// LS Electric XG5000 project: 과년68_2_3
// PLC NewPLC
// module base 0 slot 0: 입출력 모듈:XBC-DR20S (DC 24V 입력 12점, 릴레이 출력 8점)

PROGRAM NewProgram (task: 스캔 프로그램)

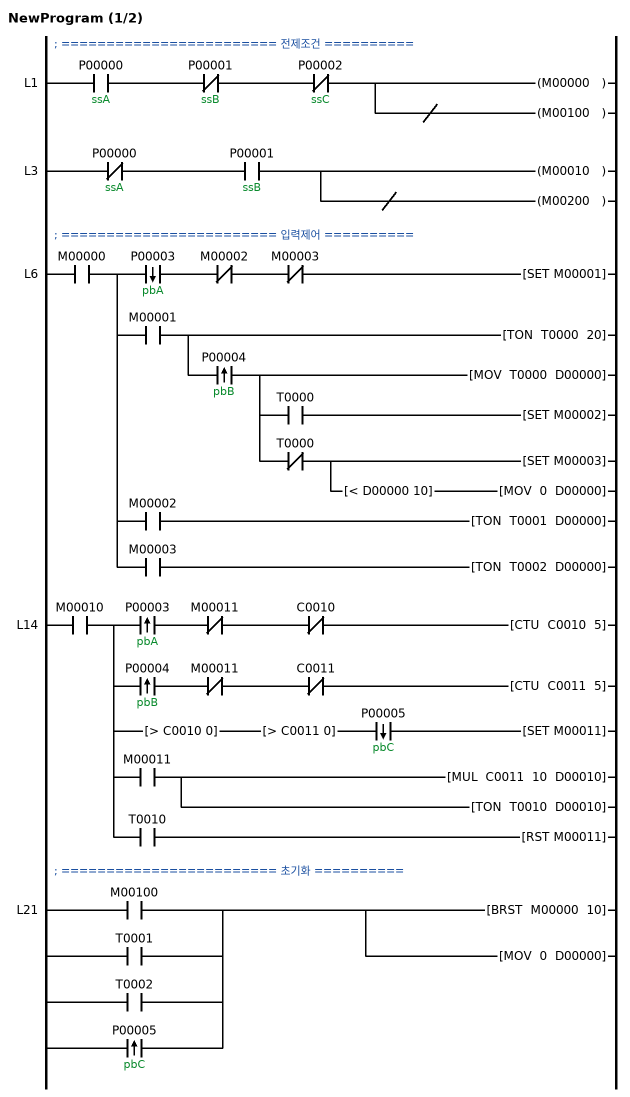
// ======================== 전제조건 ==========
; L1
LOAD      P00000	// ssA
AND NOT   P00001	// ssB
AND NOT   P00002	// ssC
OUT       M00000
NOT
OUT       M00100
; L3
LOAD NOT  P00000	// ssA
AND       P00001	// ssB
OUT       M00010
NOT
OUT       M00200
// ======================== 입력제어 ==========
; L6
LOAD      M00000
MPUSH
ANDN      P00003	// pbA
AND NOT   M00002
AND NOT   M00003
SET       M00001
MLOAD
AND       M00001
TON       T0000 20
ANDP      P00004	// pbB
MOV       T0000 D00000
MPUSH
AND       T0000
SET       M00002
MPOP
AND NOT   T0000
SET       M00003
AND<      D00000 10
MOV       0 D00000
MLOAD
AND       M00002
TON       T0001 D00000
MPOP
AND       M00003
TON       T0002 D00000
; L14
LOAD      M00010
MPUSH
ANDP      P00003	// pbA
AND NOT   M00011
AND NOT   C0010
CTU       C0010 5
MLOAD
ANDP      P00004	// pbB
AND NOT   M00011
AND NOT   C0011
CTU       C0011 5
MLOAD
AND>      C0010 0
AND>      C0011 0
ANDN      P00005	// pbC
SET       M00011
MLOAD
AND       M00011
MUL       C0011 10 D00010
TON       T0010 D00010
MPOP
AND       T0010
RST       M00011
// ======================== 초기화 ==========
; L21
LOAD      M00100
OR        T0001
OR        T0002
ORP       P00005	// pbC
BRST      M00000 10
MOV       0 D00000

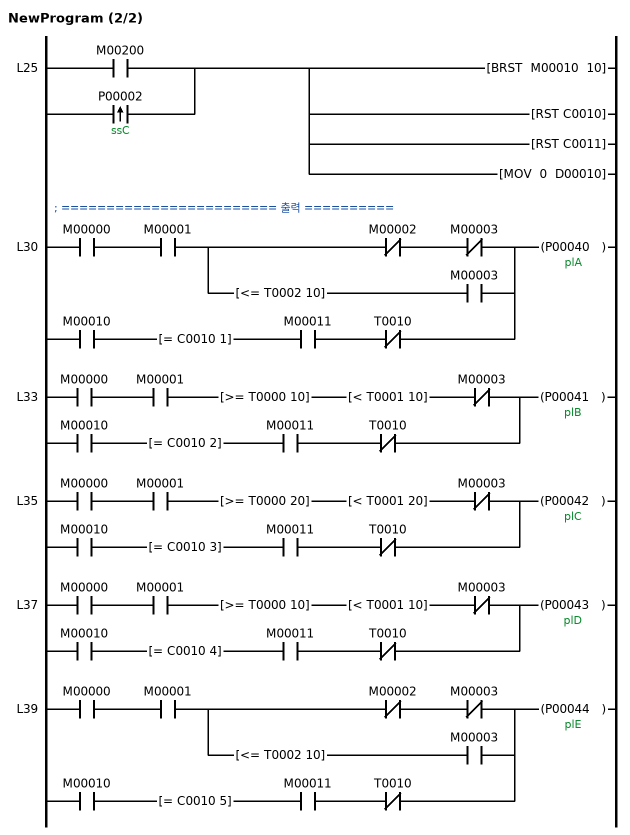
; L25
LOAD      M00200
ORP       P00002	// ssC
BRST      M00010 10
RST       C0010
RST       C0011
MOV       0 D00010
// ======================== 출력 ==========
; L30
LOAD      M00000
AND       M00001
LOAD NOT  M00002
AND NOT   M00003
LOAD<=    T0002 10
AND       M00003
OR LOAD
AND LOAD
LOAD      M00010
AND=      C0010 1
AND       M00011
AND NOT   T0010
OR LOAD
OUT       P00040	// plA
; L33
LOAD      M00000
AND       M00001
AND>=     T0000 10
AND<      T0001 10
AND NOT   M00003
LOAD      M00010
AND=      C0010 2
AND       M00011
AND NOT   T0010
OR LOAD
OUT       P00041	// plB
; L35
LOAD      M00000
AND       M00001
AND>=     T0000 20
AND<      T0001 20
AND NOT   M00003
LOAD      M00010
AND=      C0010 3
AND       M00011
AND NOT   T0010
OR LOAD
OUT       P00042	// plC
; L37
LOAD      M00000
AND       M00001
AND>=     T0000 10
AND<      T0001 10
AND NOT   M00003
LOAD      M00010
AND=      C0010 4
AND       M00011
AND NOT   T0010
OR LOAD
OUT       P00043	// plD
; L39
LOAD      M00000
AND       M00001
LOAD NOT  M00002
AND NOT   M00003
LOAD<=    T0002 10
AND       M00003
OR LOAD
AND LOAD
LOAD      M00010
AND=      C0010 5
AND       M00011
AND NOT   T0010
OR LOAD
OUT       P00044	// plE